PROGRAM MAIN
VAR
	iWatchdog:UDINT;//The watchdog variable name written to by the remote plc

	fbLogHandler: FB_LogHandler;
END_VAR

(*Ethercat Diagnostics*)
//DIAGNOSTICS();



(* Call all Programs*)
PRG_ILK();
PRG_GEM1_DIFF_PUMP();
PRG_GEM2_DIFF_PUMP();
PRG_ROOTS();
PRG_GATT();
PRG_GEM1();
PRG_GEM2();
PRG_PMPS();
//Log Handler
fbLogHandler();

END_PROGRAM

(* stored: Version 1.1.0.1, ProductVersion 3.1.4022.18
   POU MAIN: Id {08fcf07b-a57e-4f6f-85ed-e3315e0ea5b4}, SpecialFunc None *)
